PROGRAM MAIN
VAR
END_VAR

END_PROGRAM

(* stored: Version 1.1.0.1, ProductVersion 3.1.0.38
   POU MAIN: Id {26474e12-5de3-4ee8-b8b8-363965c8c934}, SpecialFunc None *)
